{attribute 'GeneratedUsingTerminal: EL3681-0000-0018'}
{attribute addProperty BoxType "EL3681-0000-0018"}
{attribute addProperty Id "ControlAT %Q*Control_18D542D94"}
{attribute addProperty CRC "706248645"}
{attribute addProperty Size "4"}
TYPE SAI_Range_2A187FC5 :
STRUCT
	{attribute addProperty Name "Control"}
	Control AT %Q* : Control_18D542D9;
END_STRUCT
END_TYPE

(* stored: Version 1.2.0.0, ProductVersion 3.1.4024.9
   DUT SAI_Range_2A187FC5: Id {6e903d79-bd4e-4d3e-8839-107e6a853b50} *)
